Staubli VAL3: check_solid.dtx

mdesc mNomSpeed
bool bCreate_cube
bool bCreate_cylind
bool bCreate_plane
bool bCreate_sphere
frame fPlane = {fatherId=world[0]}
pointRx pOrigin_sphere = {fatherId=world[0]}
num nRadius_sphere
frame fCube = {fatherId=world[0]}
num nDistanceX_cube
num nDistanceY_cube
num nDistanceZ_cube
frame fCylinder = {fatherId=world[0]}
num nRadius_cyl
num nDistanceZ_cyl
pointRx pOrigin_cylind = {fatherId=world[0]}
